TYPE Eh_ErrorEntry_typ:
STRUCT
	SourceId		: UDINT;
	SubSourceId		: UDINT;
	ErrorId			: UDINT;
	ErrorText		: STRING(500);
	MotorEvents		: enumMotorEvents;	
END_STRUCT
END_TYPE

(* stored: Version 1.1.0.1, ProductVersion 3.1.4024.3
   DUT Eh_ErrorEntry_typ: Id {e5f8aba5-7785-0212-0240-7e6debb9c5a4} *)
